SUBAPPLICATION SubApp_PC_A (* Geraet A (Station 11, 192.168.1.11): 2 VT-SoftKeys (Softkey_IXA, F1=Hoch/F2=Runter) statt physischer logiBUS_IXA-Eingaenge wie in Training_10 - schreiben aktiv per OPC-UA (CLIENT_1_0) auf die von Geraet B ueberwachten Knoten. Zusaetzlich GreenWhiteBackground je Taste: faerbt den jeweiligen SoftKey nach dem von Geraet B lokal ueberwachten, TATSAECHLICH erreichten Zustand (nach ILOCK-Arbitrierung/Schutzzeit), nicht nach dem rohen Tastendruck - 'SUB style', das Protokoll steckt im FB-Netz dieses Composites, nicht in der Resource des Geraets. Softkey_IXA liest kontinuierlich (wie logiBUS_IXA), kein REQ-Polling noetig - INIT (EInit) startet die Ueberwachung automatisch, analog zum Vorbild Softkey_IXA_TO_logiBUS_QXA_BG.SUB. *)
  (* Standard: 61499-2; Description: Copyright (c) 2026 Meisterschulen am Ostbahnhof This program and the accompanying materials are made available under the terms of the Eclipse Public License 2.0 which is available at https://www.eclipse.org/legal/epl-2.0/ SPDX-License-Identifier: EPL-2.0 *)
  (* Version 1.0, 2026-09-05, Franz Höpfinger, Meisterschulen am Ostbahnhof, initial API and implementation and/or initial documentation *)
  PACKAGE subapp::Training_11_OPC_UA_RES;
  IMPORT Uebungen::const::UT::DefaultPool::SoftKey_F1;
  IMPORT Uebungen::const::UT::DefaultPool::SoftKey_F2;
  IMPORT VV::const::OPC_UA::myOpcUaAddresses::SW1_UP_REMOTE_WRITE;
  IMPORT VV::const::OPC_UA::myOpcUaAddresses::SW1_DOWN_REMOTE_WRITE;
  IMPORT VV::const::OPC_UA::myOpcUaAddresses::SW1_UP_STATE_LOCAL_READ;
  IMPORT VV::const::OPC_UA::myOpcUaAddresses::SW1_DOWN_STATE_LOCAL_READ;
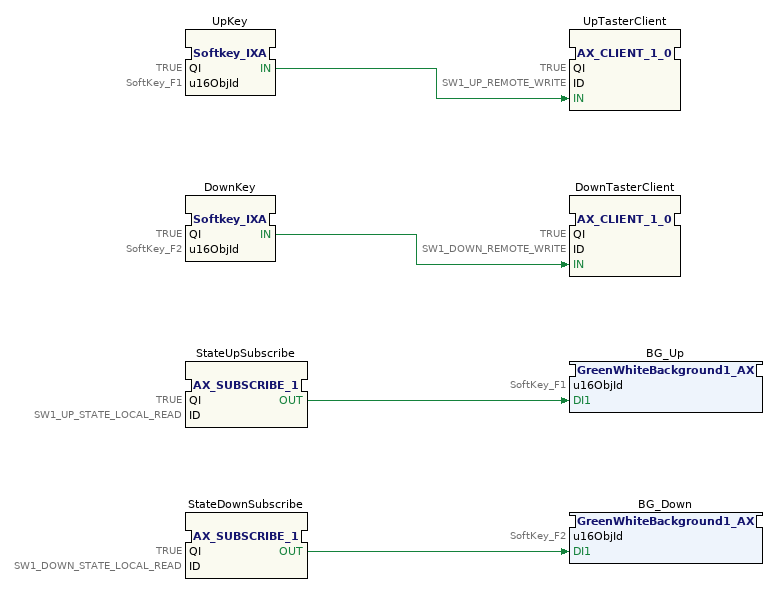
  FBS
    UpKey : isobus::UT::io::Softkey::Softkey_IXA(QI := TRUE, u16ObjId := SoftKey_F1);
    DownKey : isobus::UT::io::Softkey::Softkey_IXA(QI := TRUE, u16ObjId := SoftKey_F2);
    UpTasterClient : adapter::net::AX_CLIENT_1_0(QI := TRUE, ID := SW1_UP_REMOTE_WRITE);
    DownTasterClient : adapter::net::AX_CLIENT_1_0(QI := TRUE, ID := SW1_DOWN_REMOTE_WRITE);
    StateUpSubscribe : adapter::net::AX_SUBSCRIBE_1(QI := TRUE, ID := SW1_UP_STATE_LOCAL_READ);
    StateDownSubscribe : adapter::net::AX_SUBSCRIBE_1(QI := TRUE, ID := SW1_DOWN_STATE_LOCAL_READ);
  END_FBS
  SUBAPPS
    BG_Up : MyLib::sys::GreenWhiteBackground1_AX(u16ObjId := SoftKey_F1);
    BG_Down : MyLib::sys::GreenWhiteBackground1_AX(u16ObjId := SoftKey_F2);
  END_SUBAPPS
  ADAPTER_CONNECTIONS
    UpKey.IN TO UpTasterClient.IN;
    DownKey.IN TO DownTasterClient.IN;
    StateUpSubscribe.OUT TO BG_Up.DI1;
    StateDownSubscribe.OUT TO BG_Down.DI1;
  END_CONNECTIONS
END_SUBAPPLICATION
